TYPE ST_PROCESS_DATA :
STRUCT
  nProcessId          : e_instance; // target process
  {attribute 'displaymode':='bin'}
  wTarget             : T_PROCESS;  // where and how many stations are to be used in process
END_STRUCT
END_TYPE

(* stored: Version 1.1.0.1
   DUT ST_PROCESS_DATA: Id {a3bf93e1-2773-4ab2-bd47-0b7a8158d7ce} *)
